FUNCTION FC_OvrManagement : UINT
VAR_INPUT
	X_min 			: UINT;
    X_max 			: UINT;
    Y_min 			: UINT;
    Y_max 			: UINT;
	Counter			: UINT;
	SetCounterDone 	: BOOL;
END_VAR
VAR_OUTPUT
	SetCounte 		: BOOL;
	SetCounteValue 	: UINT;
END_VAR

IF NOT SetCounterDone THEN
	IF Counter < X_min THEN
		SetCounteValue := X_min;
		SetCounte := TRUE;
	ELSIF Counter > X_max THEN
		SetCounteValue := X_max;
		SetCounte := TRUE;
	ELSE
		FC_OvrManagement := (((Counter - X_min) * (Y_max - Y_min)) / (X_max - X_min) + Y_min);
	END_IF
ELSIF SetCounte THEN
	SetCounte := FALSE;
END_IF

END_FUNCTION

(* stored: Version 1.1.0.1, ProductVersion 3.1.4024.13
   POU FC_OvrManagement: Id {0b599ed5-89b6-46bd-b89a-4a3bc38be01e}, SpecialFunc None *)
